(* IEC 61131-3 sources: plc-modbus-safety-controller/plc, 2 files *)

(* ---- ModbusGateway.st ---- *)
FUNCTION_BLOCK FB_ModbusGateway
VAR_INPUT
    StateCode : USINT;
    FaultActive : BOOL;
    GuardClosed : BOOL;
    PressureHealthy : BOOL;
    EmergencyStop : BOOL;
    CommandRegister : UINT;
END_VAR
VAR_OUTPUT
    StateRegister : UINT;
    SafetyRegister : UINT;
    AcceptedCommand : UINT;
END_VAR

StateRegister := UINT(StateCode);
SafetyRegister := 0;
IF GuardClosed THEN SafetyRegister := SafetyRegister OR 1; END_IF;
IF PressureHealthy THEN SafetyRegister := SafetyRegister OR 2; END_IF;
IF EmergencyStop THEN SafetyRegister := SafetyRegister OR 4; END_IF;
IF FaultActive THEN SafetyRegister := SafetyRegister OR 8; END_IF;

IF CommandRegister <= 3 THEN
    AcceptedCommand := CommandRegister;
ELSE
    AcceptedCommand := 0;
END_IF;
END_FUNCTION_BLOCK

(* ---- MotorController.st ---- *)
TYPE E_MotorState :
(
    stopped,
    starting,
    running,
    stopping,
    tripped
);
END_TYPE

FUNCTION_BLOCK FB_MotorController
VAR_INPUT
    StartCommand : BOOL;
    StopCommand : BOOL;
    ResetCommand : BOOL;
    EmergencyStop : BOOL;
    GuardClosed : BOOL;
    PressureHealthy : BOOL;
    Overload : BOOL;
    NowMs : UDINT;
    StartDelayMs : UDINT := 1500;
    StopDelayMs : UDINT := 800;
END_VAR
VAR_OUTPUT
    State : E_MotorState := stopped;
    RunOutput : BOOL;
    FaultActive : BOOL;
    TransitionSequence : UDINT;
END_VAR
VAR
    StateSinceMs : UDINT;
    Unsafe : BOOL;
END_VAR

Unsafe := EmergencyStop OR NOT GuardClosed OR NOT PressureHealthy OR Overload;

IF Unsafe THEN
    IF State <> tripped THEN
        State := tripped;
        StateSinceMs := NowMs;
        TransitionSequence := TransitionSequence + 1;
    END_IF;
ELSIF State = tripped THEN
    IF ResetCommand THEN
        State := stopped;
        StateSinceMs := NowMs;
        TransitionSequence := TransitionSequence + 1;
    END_IF;
ELSIF State = stopped AND StartCommand THEN
    State := starting;
    StateSinceMs := NowMs;
    TransitionSequence := TransitionSequence + 1;
ELSIF State = starting AND StopCommand THEN
    State := stopping;
    StateSinceMs := NowMs;
    TransitionSequence := TransitionSequence + 1;
ELSIF State = starting AND (NowMs - StateSinceMs) >= StartDelayMs THEN
    State := running;
    StateSinceMs := NowMs;
    TransitionSequence := TransitionSequence + 1;
ELSIF State = running AND StopCommand THEN
    State := stopping;
    StateSinceMs := NowMs;
    TransitionSequence := TransitionSequence + 1;
ELSIF State = stopping AND (NowMs - StateSinceMs) >= StopDelayMs THEN
    State := stopped;
    StateSinceMs := NowMs;
    TransitionSequence := TransitionSequence + 1;
END_IF;

FaultActive := State = tripped;
RunOutput := State = running;
END_FUNCTION_BLOCK
